INTERFACE I_EncoderScaling

PROPERTY EncoderCount : UDINT
GET
END_GET
END_PROPERTY

METHOD EncoderScaling : UDINT
END_METHOD

END_INTERFACE

(* stored: Version 1.1.0.1
   Itf I_EncoderScaling: Id {22b9eaa5-9d83-47ac-afe3-1fbdad58c443}
   Property EncoderCount: Id {93445dbc-b389-4916-96fe-856216773594}
   Get Get: Id {34af533c-cf5f-4a77-a012-16b3af7602a0}
   Method EncoderScaling: Id {aa4aa2b3-d892-434a-940d-c34b50da3016} *)
